{attribute addProperty BoxType "CU1123-0000-0016"}
{attribute addProperty Id "A_0002_CU1123_0010_0016A_0002_CU1123_0010_0016_C16CD0B3950118.75"}
{attribute addProperty CRC "2833566819"}
{attribute addProperty SizeInBites "950"}
{attribute addProperty SizeInBytes "118.75"}
TYPE A_0001_CU1123_0000_0016_A8E4CC63 EXTENDS CU1123_179A0949 :
STRUCT
	{attribute addProperty Name "A_0002_CU1123_0010_0016"}
	A_0002_CU1123_0010_0016 : A_0002_CU1123_0010_0016_C16CD0B3;
END_STRUCT
END_TYPE

(* stored: Version 1.2.0.0, ProductVersion 3.1.4024.9
   DUT A_0001_CU1123_0000_0016_A8E4CC63: Id {0312027e-6afe-416d-a472-ffbb65312a27} *)
